{attribute 'GeneratedUsingTerminal: EK1100-0000-0018'}
{attribute addProperty BoxType "EK1100-0000-0018"}
{attribute addProperty Id "Beckhoff_ER1xxxEK1122Beckhoff_ER1xxxEK1122_0C0834C7508"}
{attribute addProperty CRC "1820564652"}
{attribute addProperty Size "508"}
TYPE Beckhoff_ER1xxx_6C839CAC EXTENDS EK1100_AB5A9467 :
STRUCT
	{attribute addProperty Name "Beckhoff_ER1xxxEK1122"}
	Beckhoff_ER1xxxEK1122 : Beckhoff_ER1xxxEK1122_0C0834C7;
END_STRUCT
END_TYPE

(* stored: Version 1.2.0.0, ProductVersion 3.1.4024.9
   DUT Beckhoff_ER1xxx_6C839CAC: Id {1245ad83-ee77-4285-958b-40a27c13b026} *)
